PROGRAM MAIN
VAR
END_VAR

END_PROGRAM

(* stored: Version 1.1.0.1
   POU MAIN: Id {29889874-30b4-4503-8dfb-8ef77ee8e328} *)
